PROGRAM MAIN
VAR
	fbMC_Power1: MC_Power;
	xEnable: BOOL;
	xControlPower: BOOL;
	fbMC_Power2: MC_Power;
	lrAxis2_Override: LREAL;
	fmMC_Reset1: MC_Reset;
	xAxisReset: BOOL;
	fmMC_Reset2: MC_Reset;
	Axis: INT;
	Execute: INT;
	xMachineReset: BOOL;
	fbMC_MoveRelative1: MC_MoveRelative;
	xExecuteDistance: BOOL;
	lrDistance: LREAL := 10.0;
	fbMC_MoveAbsolute1: MC_MoveAbsolute;
	xExecuteMoveAbsolute1: BOOL;
	lrPosition: LREAL;
	fbMC_MoveVelocity1: MC_MoveVelocity;
	xExecuteVelo: BOOL;
	fbMC_Halt1: MC_Halt;
	xExecuteHalt1: BOOL;
	fbMC_Stop1: MC_Stop;
	xExecuteStop1: BOOL;
	fbMC_MoveMod: MC_MoveModulo;
	xExecuteMoveMod1: BOOL;
	lrPosMod: LREAL;
	fb_MC_Jog_StandardSLow1: MC_Jog;
	xJogFwdStandardSlow: BOOL;
	xJogBckwdStandardSlow: BOOL;
END_VAR

GVL.Axis1.ReadStatus();
GVL.Axis2.ReadStatus();

IF xControlPower THEN
	xEnable := TRUE;
ELSE
	xEnable := FALSE;
END_IF
fbMC_Power1(
		Axis:= GVL.Axis1, 
		Enable:= xEnable, 
		Enable_Positive:= xEnable, 
		Enable_Negative:= xEnable, 
		Override:= 100.0 
		);
		
fbMC_Power2(
	Axis:= GVL.Axis2, 
	Enable:= xEnable, 
	Enable_Positive:= xEnable, 
	Enable_Negative:= xEnable, 
	Override:= lrAxis2_Override 
	);
	
	IF xMachineReset THEN
		xAxisReset := TRUE;
	ELSE 
		xAxisReset := FALSE;
	END_IF
	
fbMC_MoveRelative1(
	Axis:= GVL.Axis1, 
	Execute:= xExecuteDistance, 
	Distance:= lrDistance, 
	Velocity:= 5.0 
 );
	
fbMC_MoveAbsolute1(
	Axis:= GVL.Axis1, 
	Execute:= xExecuteMoveAbsolute1, 
	Position:= lrPosition, 
	Velocity:= 50.0 
 );

fbMC_MoveVelocity1(
	Axis:= GVL.Axis1, 
	Execute:= xExecuteVelo, 
	Velocity:= 25, 
	 );

fbMC_Halt1(
	Axis:= GVL.Axis1, 
	Execute:= xExecuteHalt1 );

fbMC_Stop1(
	Axis:= GVL.Axis1, 
	Execute:=  xExecuteStop1
 );


fbMC_MoveMod(
	Axis:= GVL.Axis1, 
	Execute:= xExecuteMoveMod1, 
	Position:= lrPosMod, 
	Velocity:= 25.0, 
 	Direction:= MC_Direction.MC_Positive_Direction
 );

E_JogMode.MC_JOGMODE_STANDARD_SLOW;
E_JogMode.MC_JOGMODE_STANDARD_FAST;
E_JogMode.MC_JOGMODE_CONTINOUS;
E_JogMode.MC_JOGMODE_INCHING;
E_JogMode.MC_JOGMODE_INCHING_MODULO;

fb_MC_Jog_StandardSLow1(
	Axis:= GVL.Axis1, 
	JogForward:= xJogFwdStandardSlow,
	JogBackwards:= xJogBckwdStandardSlow, 
	Mode:= E_JogMode.MC_JOGMODE_STANDARD_SLOW 
 );


fmMC_Reset1(
		Axis:= GVL.Axis1, 
		Execute:= xAxisReset AND GVL.Axis1.Status.Error
		);
	
fmMC_Reset2(
		Axis:= GVL.Axis2, 
		Execute:= xAxisReset AND GVL.Axis2.Status.Error
		);

END_PROGRAM

(* stored: Version 1.1.0.1, ProductVersion 3.1.4024.12
   POU MAIN: Id {15633034-a0d2-44bd-a0e3-22c18de57c41}, SpecialFunc None *)
